// TIA Portal V16 export
// export: Created 2019-09-22T11:06:18.1471742Z, ExportSetting WithDefaults, DisplayName Totally Integrated Automation Portal, DisplayVersion V16, DisplayName TIA Portal Version Control Interface, DisplayVersion V16, DisplayName TIA Portal Openness, DisplayVersion V16, DisplayName STEP 7 Professional, DisplayVersion V16, DisplayName SIMATIC Energy Suite, DisplayVersion V16, DisplayName STEP 7 Safety, DisplayVersion V16, DisplayName WinCC Professional, DisplayVersion V16, DisplayName SIMATIC Visualization Architect, DisplayVersion V16
ORGANIZATION_BLOCK "Startup"   // OB100, FBD, Startup
TITLE = "Complete Restart"
{ S7_Optimized_Access := 'TRUE' }
VERSION : 0.1
// //============================================================================
// //SIEMENS AG
// //(c)Copyright 2015 All Rights Reserved
// //-----------------------------------------------------------------------------
// //Library: -
// //Tested with: S7-1516-3 PN/DP FW 1.7
// //Engineering: TIA Portal V13 SP1
// //Restrictions: -
// //Requirements: -
// //Functionality: Startup OB for Configuration control and Diagnostic
// //-----------------------------------------------------------------------------
// //Change log table:
// //Version  Date       Expert in charge Changes applied
// //01.00.00 24.03.2015 Siemens Industry Online Support First released version
// //============================================================================
// stored: AutoNumber true, IsIECCheckEnabled false, SetENOAutomatically false
   VAR_INPUT
      LostRetentive : Bool;   // True if retentive data are lost
      LostRTC : Bool;   // True if date and time are lost
   END_VAR
BEGIN

REGION Network 1: call startup and diagnostic of PLC
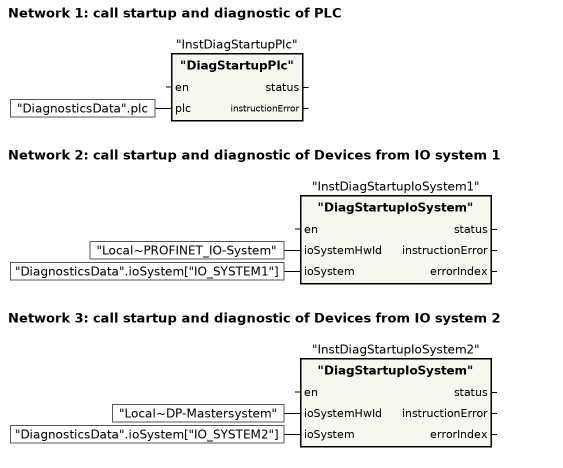
   "InstDiagStartupPlc"(plc := "DiagnosticsData".plc);   // "DiagStartupPlc"
END_REGION

REGION Network 2: call startup and diagnostic of Devices from IO system 1
   "InstDiagStartupIoSystem1"(ioSystemHwId := "Local~PROFINET_IO-System",   // "DiagStartupIoSystem"
                           ioSystem := "DiagnosticsData".ioSystem["IO_SYSTEM1"]);
END_REGION

REGION Network 3: call startup and diagnostic of Devices from IO system 2
   "InstDiagStartupIoSystem2"(ioSystemHwId := "Local~DP-Mastersystem",   // "DiagStartupIoSystem"
                           ioSystem := "DiagnosticsData".ioSystem["IO_SYSTEM2"]);
END_REGION
END_ORGANIZATION_BLOCK
